(* IEC 61131-3 sources: volt/packages/volt-lsp-iec/test-corpus/awa-palletizer/Device/Plc Logic/Application/Library Manager/Component Manager, 29 files *)

(* ---- EVTPARAM_CMPMGR_DISABLEOPERATION.dut ---- *)
TYPE EVTPARAM_CMPMGR_DISABLEOPERATION :
STRUCT
	UDICMPID : UDINT;
	UDIOPERATION : UDINT;
	UDICMPIDDISABLED : UDINT;
	BDISABLE : DINT;
END_STRUCT
END_TYPE

(* ---- EVTPARAM_CMPMGR_LICENSEREQUEST.dut ---- *)
TYPE EVTPARAM_CMPMGR_LICENSEREQUEST :
STRUCT
	ULLICENSEID : UDINT;
	ULLICENSEVALUE : UDINT;
END_STRUCT
END_TYPE

(* ---- EVTPARAM_CMPMGR_LICENSESTATE.dut ---- *)
TYPE EVTPARAM_CMPMGR_LICENSESTATE :
STRUCT
	MULFIRMCODE : UDINT;
	MULPRODUCTCODE : UDINT;
	MULFEATUREMAP : UDINT;
	PSZLICENSENAME : POINTER TO STRING;
	STATE : RUNTIME_LICENSE_STATE;
	SECONDSTOEXPIRATION : UDINT;
	ERRORCODE : RTS_IEC_RESULT;
END_STRUCT
END_TYPE

(* ---- EVTPARAM_CMPMGR_PREPAREEXITCOMMPROCESSING.dut ---- *)
TYPE EVTPARAM_CMPMGR_PREPAREEXITCOMMPROCESSING :
STRUCT
	BLASTCALL : DINT;
	BFURTHERCALLNECESSARY : DINT;
END_STRUCT
END_TYPE

(* ---- EVTPARAM_CMPMGR_SHUTDOWN.dut ---- *)
TYPE EVTPARAM_CMPMGR_SHUTDOWN :
STRUCT
	PDUMMY : POINTER TO BYTE;
END_STRUCT
END_TYPE

(* ---- LICENSEFUNCTIONS.dut ---- *)
TYPE LICENSEFUNCTIONS :
STRUCT
	DWSTRUCTSIZE : DWORD;
	PFGETUSERLICENSEVALUE : POINTER TO BYTE;
	PFCONFDYNLICCHALLENGE : POINTER TO BYTE;
	PFREQDYNLICCHALLENGE : POINTER TO BYTE;
	DWVERSION : DWORD;
END_STRUCT
END_TYPE

(* ---- RUNTIME_LICENSE_STATE.dut ---- *)
TYPE RUNTIME_LICENSE_STATE :
(
	INIT := 0,
	DEMOMODE := 1,
	LICENSED := 2,
	LICENSE_LOST := 3,
	TRIGGER_SHUTDOWN := 4,
	SAFEMODE := 5
);
END_TYPE

(* ---- COMPONENTID.gvl ---- *)
VAR_GLOBAL
	CMPID_CMPMGR : DWORD := 16#1;
	CMPID_IECCODE : DWORD := 16#1000;
	CMPID_CMPFILETRANSFER : DWORD := 16#5E;
END_VAR

(* ---- EVENTIDS.gvl ---- *)
VAR_GLOBAL
	EVTPARAMID_CMPMGR_SHUTDOWN : WORD := 16#1;
	EVTVERSION_CMPMGR_SHUTDOWN : WORD := 16#1;
	EVTPARAMID_CMPMGR_DISABLEOPERATION : WORD := 16#2;
	EVTVERSION_CMPMGR_DISABLEOPERATION : WORD := 16#1;
	EVTPARAMID_CMPMGR_PREPAREEXITCOMMPROCESSING : WORD := 16#3;
	EVTVERSION_CMPMGR_PREPAREEXITCOMMPROCESSING : WORD := 16#1;
	EVTPARAMID_CMPMGR_LICENSEREQUEST : WORD := 16#4;
	EVTVERSION_CMPMGR_LICENSEREQUEST : WORD := 16#1;
	EVTPARAMID_CMPMGR_LICENSE_STATE : WORD := 16#5;
	EVTVERSION_CMPMGR_LICENSE_STATE : WORD := 16#1;
	EVT_CMPMGR_PREPARESHUTDOWN : DWORD := 16#10001;
	EVT_CMPMGR_PREPAREEXITCOMM : DWORD := 16#10002;
	EVT_CMPMGR_PREPAREEXITTASKS : DWORD := 16#10003;
	EVT_CMPMGR_DISABLEOPERATION : DWORD := 16#10006;
	EVT_CMPMGR_PREPAREEXITCOMMPROCESSING : DWORD := 16#10007;
	EVT_CMPMGR_LICENSEREQUEST : DWORD := 16#10008;
	EVT_CMPMGR_LICENSESTATE : DWORD := 16#10009;
END_VAR

(* ---- OPERATIONS.gvl ---- *)
VAR_GLOBAL
	OP_FILE_TRANSFER_DOWNLOAD : DWORD := 1;
	OP_FILE_TRANSFER_UPLOAD : DWORD := 2;
END_VAR

(* ---- CMADDCOMPONENT.pou ---- *)
FUNCTION CMADDCOMPONENT : RTS_IEC_HANDLE
VAR_INPUT
	PSZCOMPONENT : REFERENCE TO STRING;
	UDICMPID : UDINT;
	UDIVERSION : UDINT;
	PRESULT : POINTER TO RTS_IEC_RESULT;
END_VAR
END_FUNCTION

(* ---- CMADDCOMPONENT2.pou ---- *)
FUNCTION CMADDCOMPONENT2 : RTS_IEC_HANDLE
VAR_INPUT
	PSZCOMPONENT : REFERENCE TO STRING;
	UDIVERSION : UDINT;
	UDICMPID : POINTER TO UDINT;
	PRESULT : POINTER TO RTS_IEC_RESULT;
END_VAR
END_FUNCTION

(* ---- CMEXITCOMPONENT.pou ---- *)
FUNCTION CMEXITCOMPONENT : RTS_IEC_RESULT
VAR_INPUT
	HCOMPONENT : RTS_IEC_HANDLE;
END_VAR
END_FUNCTION

(* ---- CMGETCOMPONENTBYNAME.pou ---- *)
FUNCTION CMGETCOMPONENTBYNAME : RTS_IEC_HANDLE
VAR_INPUT
	PSZCOMPONENT : REFERENCE TO STRING;
	PRESULT : POINTER TO RTS_IEC_RESULT;
END_VAR
END_FUNCTION

(* ---- CMGETCOREVERSION.pou ---- *)
FUNCTION CMGETCOREVERSION : RTS_IEC_RESULT
VAR_INPUT
	PUDICOREVERSION : POINTER TO UDINT;
END_VAR
END_FUNCTION

(* ---- CMINITCOMPONENT.pou ---- *)
FUNCTION CMINITCOMPONENT : RTS_IEC_RESULT
VAR_INPUT
	HCOMPONENT : RTS_IEC_HANDLE;
END_VAR
END_FUNCTION

(* ---- CMREGISTERGETUSERLICENSEVALUE.pou ---- *)
FUNCTION CMREGISTERGETUSERLICENSEVALUE : RTS_IEC_RESULT
VAR_INPUT
	PFGETUSERLICENSEVALUE : POINTER TO BYTE;
END_VAR
END_FUNCTION

(* ---- CMREGISTERLICENSEFUNCTIONS.pou ---- *)
FUNCTION CMREGISTERLICENSEFUNCTIONS : RTS_IEC_RESULT
VAR_INPUT
	LICENSEFUNCTIONS : LicenseFunctions;
END_VAR
END_FUNCTION

(* ---- CMREMOVECOMPONENT.pou ---- *)
FUNCTION CMREMOVECOMPONENT : RTS_IEC_RESULT
VAR_INPUT
	HCOMPONENT : RTS_IEC_HANDLE;
END_VAR
END_FUNCTION

(* ---- CMSHUTDOWN.pou ---- *)
FUNCTION CMSHUTDOWN : RTS_IEC_RESULT
VAR_INPUT
	DWREASON : UDINT;
END_VAR
END_FUNCTION

(* ---- CMUNREGISTERGETUSERLICENSEVALUE.pou ---- *)
FUNCTION CMUNREGISTERGETUSERLICENSEVALUE : RTS_IEC_RESULT
VAR_INPUT
	PFGETUSERLICENSEVALUE : POINTER TO BYTE;
END_VAR
END_FUNCTION

(* ---- CMUNREGISTERLICENSEFUNCTIONS.pou ---- *)
FUNCTION CMUNREGISTERLICENSEFUNCTIONS : RTS_IEC_RESULT
VAR_INPUT
	LICENSEFUNCTIONS : LicenseFunctions;
END_VAR
END_FUNCTION

(* ---- CMUTLCWSTRCPY.pou ---- *)
FUNCTION CMUTLCWSTRCPY : RTS_IEC_RESULT
VAR_INPUT
	PCWSZDEST : POINTER TO RTS_IEC_CWCHAR;
	NDESTSIZE : __XINT;
	PCWSZSRC : POINTER TO RTS_IEC_CWCHAR;
END_VAR
END_FUNCTION

(* ---- CMUTLSAFESTRCPY.pou ---- *)
FUNCTION CMUTLSAFESTRCPY : RTS_IEC_RESULT
VAR_INPUT
	PSZDEST : POINTER TO STRING(255);
	NDESTSIZE : __XINT;
	PSZSRC : POINTER TO STRING(255);
END_VAR
END_FUNCTION

(* ---- CMUTLSTRICMP.pou ---- *)
FUNCTION CMUTLSTRICMP : DINT
VAR_INPUT
	PSZSTRING1 : POINTER TO STRING;
	PSZSTRING2 : POINTER TO STRING;
END_VAR
END_FUNCTION

(* ---- CMUTLUTF8TOW.pou ---- *)
FUNCTION CMUTLUTF8TOW : RTS_IEC_RESULT
VAR_INPUT
	PUTF8STR : POINTER TO BYTE;
	UTF8BUFFERSIZE : __UXINT;
	PWSZ : POINTER TO WSTRING;
	WSTRLEN : __UXINT;
END_VAR
END_FUNCTION

(* ---- CMUTLWSTRCPY.pou ---- *)
FUNCTION CMUTLWSTRCPY : RTS_IEC_RESULT
VAR_INPUT
	PWSZDEST : POINTER TO WSTRING(255);
	NDESTSIZE : __XINT;
	PWSZSRC : POINTER TO WSTRING(255);
END_VAR
END_FUNCTION

(* ---- CMUTLWTOUTF8.pou ---- *)
FUNCTION CMUTLWTOUTF8 : RTS_IEC_RESULT
VAR_INPUT
	PWSZ : POINTER TO WSTRING;
	WSTRLEN : __UXINT;
	PUTF8STR : POINTER TO BYTE;
	UTF8BUFFERSIZE : __UXINT;
END_VAR
END_FUNCTION

(* ---- PLCOPERATIONCONTROL.pou ---- *)
FUNCTION_BLOCK PLCOPERATIONCONTROL
VAR
	_HEVENTDISABLEOPERATION : RTS_IEC_HANDLE;
	_HINTERFACEDISABLEOPERATION : RTS_IEC_HANDLE;
	_ITF : ICmpEventCallback;
	_RESULT : RTS_IEC_RESULT;
	_XDISABLEALL : BOOL;
	_XDISABLEAPPLICATIONSTOP : BOOL;
	_XDISABLEAPPLICATIONDOWNLOAD : BOOL;
	_XDISABLEAPPLICATIONONLINECHANGE : BOOL;
	_XDISABLEAPPLICATIONBP : BOOL;
	_XDISABLEAPPLICATIONFORCE : BOOL;
	_XDISABLEAPPLICATIONWRITE : BOOL;
	_XDISABLEAPPLICATIONRESET : BOOL;
	_XDISABLEAPPLICATIONSTART : BOOL;
	_XDISABLEAPPLICATIONDELETE : BOOL;
	_XDISABLEAPPLICATIONRESETORIGIN : BOOL;
	_XDISABLEFILETRANSFERUPLOAD : BOOL;
	_XDISABLEFILETRANSFERDOWNLOAD : BOOL;
	XDISABLEALL : BOOL;
	XDISABLEAPPLICATIONBREAKPOINT : BOOL;
	XDISABLEAPPLICATIONDELETE : BOOL;
	XDISABLEAPPLICATIONDOWNLOAD : BOOL;
	XDISABLEAPPLICATIONFORCE : BOOL;
	XDISABLEAPPLICATIONONLINECHANGE : BOOL;
	XDISABLEAPPLICATIONRESET : BOOL;
	XDISABLEAPPLICATIONRESETORIGIN : BOOL;
	XDISABLEAPPLICATIONSTART : BOOL;
	XDISABLEAPPLICATIONSTOP : BOOL;
	XDISABLEAPPLICATIONWRITE : BOOL;
	XDISABLEFILETRANSFERDOWNLOAD : BOOL;
	XDISABLEFILETRANSFERUPLOAD : BOOL;
END_VAR
END_FUNCTION_BLOCK

METHOD EVENTCALLBACK : UDINT
VAR_INPUT
	PEVENTPARAM : POINTER TO EventParam;
END_VAR
END_METHOD

METHOD FB_EXIT : BOOL
VAR_INPUT
	BINCOPYCODE : BOOL;
END_VAR
END_METHOD

METHOD FB_INIT : BOOL
VAR_INPUT
	BINITRETAINS : BOOL;
	BINCOPYCODE : BOOL;
END_VAR
END_METHOD
